Staubli VAL3: HMI_setValue.pgx

public program HMI_setValue(num& x_nValue, num x_nMin, num x_nMax, num x_nX, num x_nY, string& x_sItem)
  local bool l_bOk
  local bool l_bQuit
  local string l_sMessage
begin

    do
      gotoxy(x_nX,x_nY)
      put(x_sItem)
      do
        nKey=get(x_nValue)
      until nKey==270
      if x_nMin==0 and x_nMax==0
        l_bOk=true
      elseIf  x_nValue>=x_nMin and x_nValue<=x_nMax
          l_bOk=true
      else
        call language2:message(l_sMessage,38)
        popUpMsg(l_sMessage)
      endIf

    until l_bOk

    call use:nullKey(nKey)

end
